// TIA Portal V17 export
// export: Created 2024-06-16T17:47:24.0098887Z, ExportSetting WithDefaults, DisplayName Totally Integrated Automation Portal, DisplayVersion V17, DisplayName TIA Portal Openness, DisplayVersion V17, DisplayName TIA Portal Version Control Interface, DisplayVersion V17, DisplayName STEP 7 Professional, DisplayVersion V17, DisplayName STEP 7 Safety, DisplayVersion V17, DisplayName WinCC Professional, DisplayVersion V17
FUNCTION_BLOCK "Obj_St1_FB"   // FB100, FBD
{ S7_Optimized_Access := 'TRUE' }
VERSION : 0.1
// stored: AutoNumber false, IsIECCheckEnabled false, IsRetainMemResEnabled false, MemoryReserve 100, SetENOAutomatically false, UDAEnableTagReadback false
   VAR
      Axe_X : Struct
         _ActPos : Real;
         _ActVel : Real;
         _Mode : Int;
         Home : Bool;
         Halt : Bool;
         Jog : Bool;
         MoveAbs : Bool;
         MoveRel : Bool;
         MoveVel : Bool;
         PowerOff : Bool;
         PowerOn : Bool;
         SensPos : Bool;
         SensNeg : Bool;
         xBusy : Bool;
         xHomed : Bool;
         xMoveAbsDone : Bool;
         xMoveRelDone : Bool;
         xPower : Bool;
      END_STRUCT;
      Axe_Y : Struct
         _ActPos : Real;
         _ActVel : Real;
         _Mode : Int;
         Home : Bool;
         Halt : Bool;
         Jog : Bool;
         MoveAbs : Bool;
         MoveRel : Bool;
         MoveVel : Bool;
         PowerOff : Bool;
         PowerOn : Bool;
         SensPos : Bool;
         SensNeg : Bool;
         xBusy : Bool;
         xHomed : Bool;
         xMoveAbsDone : Bool;
         xMoveRelDone : Bool;
         xPower : Bool;
      END_STRUCT;
      Prehenseur_Z : Struct
         _ActPos : Real;
         _ActVel : Real;
         _Mode : Int;
         Home : Bool;
         Halt : Bool;
         Jog : Bool;
         MoveAbs : Bool;
         MoveRel : Bool;
         MoveVel : Bool;
         PowerOff : Bool;
         PowerOn : Bool;
         SensPos : Bool;
         SensNeg : Bool;
         xBusy : Bool;
         xHomed : Bool;
         xMoveAbsDone : Bool;
         xMoveRelDone : Bool;
         xPower : Bool;
      END_STRUCT;
   END_VAR
BEGIN

REGION Network 1: Station 1 - Axe X
   // //___ ModePose : 
   //          1 ---> Relative positioning
   //          2 ---> Absolute positioning
   //          3 ---> Not supported
   //          4 ---> Referencing - referencing point approach
   //          5 ---> Referencing - set referencing point
   //          6 ---> Traversing block (record mode)
   //          7 ---> Jog
   //          8 ---> Not supported
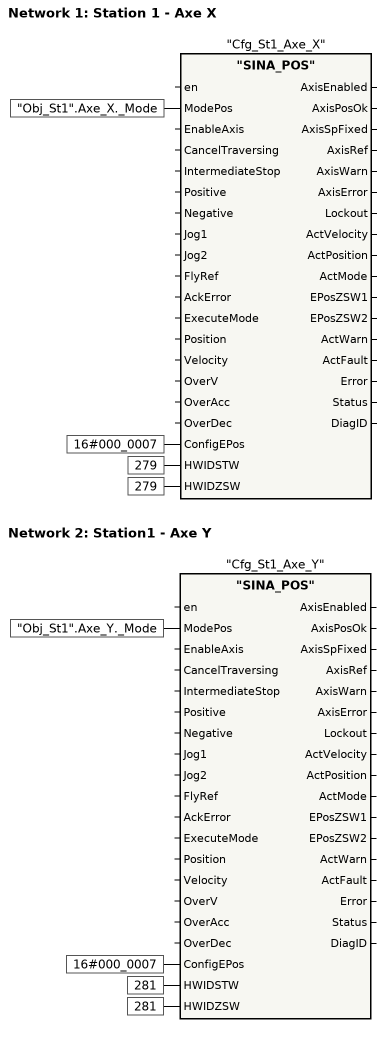
   "Cfg_St1_Axe_X"(ModePos := "Obj_St1".Axe_X._Mode, ConfigEPos := 16#000_0007, HWIDSTW := 279, HWIDZSW := 279);   // "SINA_POS"
END_REGION

REGION Network 2: Station1 - Axe Y
   // //___ ModePose : 
   //          1 ---> Relative positioning
   //          2 ---> Absolute positioning
   //          3 ---> Not supported
   //          4 ---> Referencing - referencing point approach
   //          5 ---> Referencing - set referencing point
   //          6 ---> Traversing block (record mode)
   //          7 ---> Jog
   //          8 ---> Not supported
   "Cfg_St1_Axe_Y"(ModePos := "Obj_St1".Axe_Y._Mode, ConfigEPos := 16#000_0007, HWIDSTW := 281, HWIDZSW := 281);   // "SINA_POS"
END_REGION

REGION Network 3: Station 1 - Prehenseur Z
   // //___ ModePose : 
   //          1 ---> Relative positioning
   //          2 ---> Absolute positioning
   //          3 ---> Not supported
   //          4 ---> Referencing - referencing point approach
   //          5 ---> Referencing - set referencing point
   //          6 ---> Traversing block (record mode)
   //          7 ---> Jog
   //          8 ---> Not supported
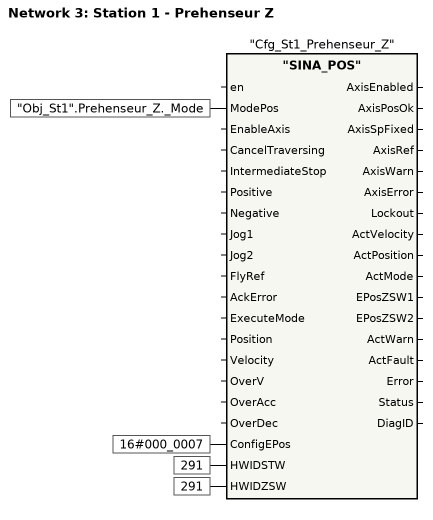
   "Cfg_St1_Prehenseur_Z"(ModePos := "Obj_St1".Prehenseur_Z._Mode,   // "SINA_POS"
                          ConfigEPos := 16#000_0007,
                          HWIDSTW := 291,
                          HWIDZSW := 291);
END_REGION
END_FUNCTION_BLOCK
